PROGRAM MAIN
VAR
	// buttons
	StartPB				: BOOL;
	StopPB				: BOOL;
	
	// sensors
	BallSensor			: BOOL;
	ColorSensor			: BOOL;
	Pusher				: BOOL;
	
	// HW outputs
	TopCylinder			: BOOL;
	BottomCylinder		: BOOL;

	// Aux. objects
	Started: BOOL;	
	DelayOn: BOOL;
	tonDelayTopCyl: TON;
	tonWhiteBall: TON;
	tonBlackBall: TON;
	tonDelay500ms: TON;
	tonPusher: TON;
END_VAR

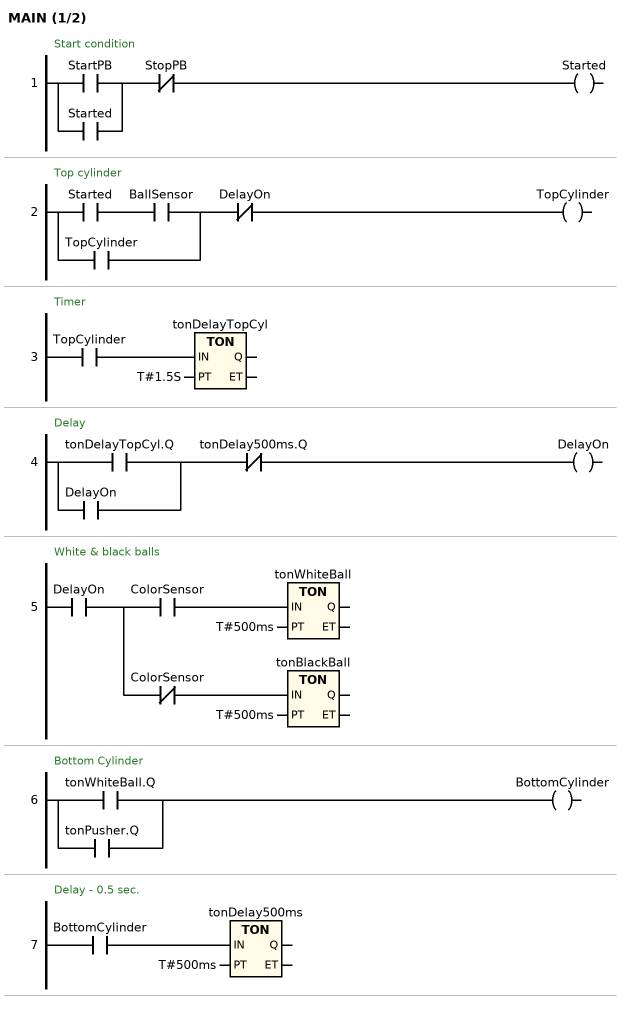
// NETWORK 1
// Start condition
Started := (StartPB OR Started) AND NOT StopPB;

// NETWORK 2
// Top cylinder
TopCylinder := (Started AND BallSensor OR TopCylinder) AND NOT DelayOn;

// NETWORK 3
// Timer
tonDelayTopCyl(IN := TopCylinder, PT := T#1.5S); // TON

// NETWORK 4
// Delay
DelayOn := (tonDelayTopCyl.Q OR DelayOn) AND NOT tonDelay500ms.Q;

// NETWORK 5
// White & black balls
tonWhiteBall(IN := DelayOn AND ColorSensor, PT := T#500ms); // TON
tonBlackBall(IN := DelayOn AND NOT ColorSensor, PT := T#500ms); // TON

// NETWORK 6
// Bottom Cylinder
BottomCylinder := tonWhiteBall.Q OR tonPusher.Q;

// NETWORK 7
// Delay - 0.5 sec.
tonDelay500ms(IN := BottomCylinder, PT := T#500ms); // TON

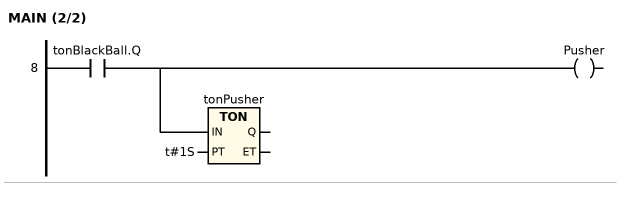
// NETWORK 8
Pusher := tonBlackBall.Q;
tonPusher(IN := tonBlackBall.Q, PT := t#1S); // TON

END_PROGRAM

(* stored: Version 1.1.0.1, ProductVersion 3.1.4024.15
   POU MAIN: Id {16e30409-2f7e-4579-a21f-682ba8e29686}, SpecialFunc None *)
